(* PLC project static_torsion.project, CODESYS CODESYS V3.5 SP17 Patch 3 *)
(* stored: creationDateTime 1970-01-01T00:00:00, modificationDateTime 2026-06-22T15:12:39.4699931 *)

FUNCTION_BLOCK ALARM
  VAR_INPUT
    xAlarmReset : BOOL;
  END_VAR
  VAR_OUTPUT
    xReady : BOOL;  (* Готовность оборудования к работе: все цепи безопасности собраны *)
    xAlarm : BOOL;
    AlarmID : INT;
  END_VAR
  VAR
    xTorqueAlarm : BOOL;
    EmergencyStop : SR;
  END_VAR

            // Оборудование готово к работе
xReady:= 	GVL.DI.CON_24V_ST AND						// цепи питание в норме
			GVL.DI.SAFE_A_ST AND						// реле безопасности A в норме
			GVL.DI.SAFE_B_ST AND						// реле безопасности B в норме
			GVL.DI.CON_220V_ST AND						// цепи управления в норме
			NOT (GVL.DI.LS_UP AND GVL.xLS_UP_EN) AND	// КВ ВЕРХ в норме или выключен флаг "КОНТРОЛИРОВАТЬ КВ ВЕРХ"
			NOT (GVL.DI.LS_DN AND GVL.xLS_DN_EN) AND	// КВ НИЗ в норме или выключен флаг "КОНТРОЛИРОВАТЬ КВ НИЗ"
			NOT (GVL.DI.LS_DOOR AND GVL.xLS_DOOR_EN);	// КВ ДВЕРЬ в норме или выключен флаг "КОНТРОЛИРОВАТЬ КВ ДВЕРЬ"

IF ABS(GVL.rTorque) > 55.0 THEN
	xTorqueAlarm := TRUE;
ELSE
	xTorqueAlarm := FALSE;
END_IF

IF GVL.DEBUG THEN
	xAlarm := FALSE;
ELSE
	EmergencyStop(SET1:= ((NOT xReady) OR xTorqueAlarm), RESET:= xAlarmReset, Q1=> xAlarm);	
END_IF
          
END_FUNCTION_BLOCK
